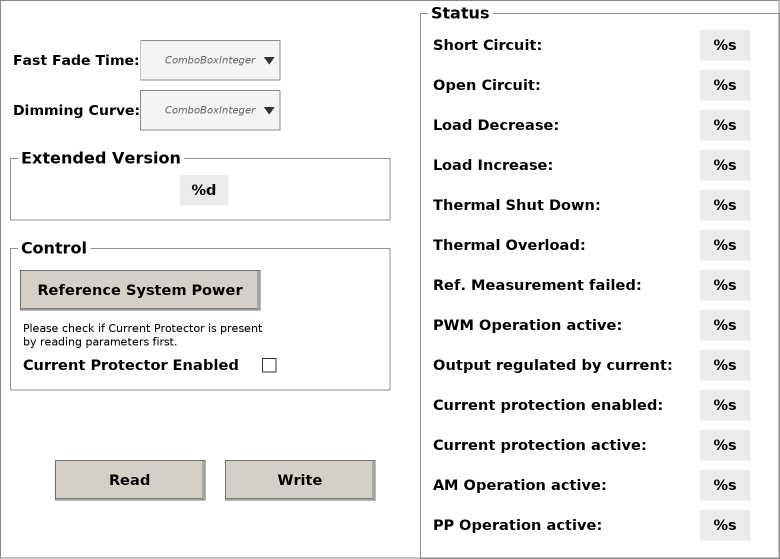
VISUALIZATION Visu_Part207Status  // 780x559
    GroupBox (420,5 360x554), "Status"
        Textfield (10,25 250x30), "Short Circuit:"
        Textfield (10,65 250x30), "Open Circuit:"
        Textfield (10,105 250x30), "Load Decrease:"
        Textfield (280,25 50x30), "%s", text variable: DALI_Commissioning.fbPart207LED.sShortCircuit
        Textfield (280,65 50x30), "%s", text variable: DALI_Commissioning.fbPart207LED.sOpenCircuit
        Textfield (280,105 50x30), "%s", text variable: DALI_Commissioning.fbPart207LED.sLoadDecrease
        Textfield (10,145 250x30), "Load Increase:"
        Textfield (280,145 50x30), "%s", text variable: DALI_Commissioning.fbPart207LED.sLoadIncrease
        Textfield (10,345 250x30), "Output regulated by current:", invisible if: DALI_Commissioning.fbPart207LED.bInvisible
        Textfield (10,385 250x30), "Current protection enabled:", invisible if: DALI_Commissioning.fbPart207LED.bInvisible
        Textfield (10,425 250x30), "Current protection active:", invisible if: DALI_Commissioning.fbPart207LED.bInvisible
        Textfield (10,185 250x30), "Thermal Shut Down:"
        Textfield (10,225 250x30), "Thermal Overload:"
        Textfield (10,265 250x30), "Ref. Measurement failed:"
        Textfield (10,465 250x30), "AM Operation active:", invisible if: DALI_Commissioning.fbPart207LED.bInvisible
        Textfield (10,505 250x30), "PP Operation active:", invisible if: DALI_Commissioning.fbPart207LED.bInvisible
        Textfield (10,305 250x30), "PWM Operation active:", invisible if: DALI_Commissioning.fbPart207LED.bInvisible
        Textfield (280,225 50x30), "%s", text variable: DALI_Commissioning.fbPart207LED.sThermalOverload
        Textfield (280,425 50x30), "%s", text variable: DALI_Commissioning.fbPart207LED.sCurrentProtectorActive, invisible if: DALI_Commissioning.fbPart207LED.bInvisible
        Textfield (280,385 50x30), "%s", text variable: DALI_Commissioning.fbPart207LED.sCurrentProtectorEnabled, invisible if: DALI_Commissioning.fbPart207LED.bInvisible
        Textfield (280,345 50x30), "%s", text variable: DALI_Commissioning.fbPart207LED.sOutputCurrentControlled, invisible if: DALI_Commissioning.fbPart207LED.bInvisible
        Textfield (280,465 50x30), "%s", text variable: DALI_Commissioning.fbPart207LED.sAMOperation, invisible if: DALI_Commissioning.fbPart207LED.bInvisible
        Textfield (280,505 50x30), "%s", text variable: DALI_Commissioning.fbPart207LED.sPowerPulseOperation, invisible if: DALI_Commissioning.fbPart207LED.bInvisible
        Textfield (280,265 50x30), "%s", text variable: DALI_Commissioning.fbPart207LED.sReferenceMeasurementFailed
        Textfield (280,185 50x30), "%s", text variable: DALI_Commissioning.fbPart207LED.sThermalShutDown
        Textfield (280,305 50x30), "%s", text variable: DALI_Commissioning.fbPart207LED.sPWMOperation, invisible if: DALI_Commissioning.fbPart207LED.bInvisible
    Button (225,460 150x40), "Write"
        OnMouseClick: execute { DALI_Commissioning.fbPart207LED.bWrite := TRUE; }
    GroupBox (10,240 380x150), "Control"
        Textfield (10,110 230x30), "Current Protector Enabled", invisible if: NOT DALI_Commissioning.fbPart207LED.bQueryCurrentProtectionDevicePresent
        Checkbox (250,110 30x30), variable: DALI_Commissioning.fbPart207LED.bCurrentProtector, invisible if: NOT DALI_Commissioning.fbPart207LED.bQueryCurrentProtectionDevicePresent, input disabled if: DALI_Commissioning.fbPart207LED.bQueryCurrentProtectionDevicePresent
        Button (10,30 240x40), "Reference System Power"
            OnMouseClick: execute { DALI_Commissioning.fbPart207LED.bReferenceSystempower := TRUE; }
        Label (10,80 300x30), "Please check if Current Protector is present by reading parameters first."
    Button (55,460 150x40), "Read"
        OnMouseClick: execute { DALI_Commissioning.fbPart207LED.bReadStatus := TRUE; }
    GroupBox (10,150 380x70), "Extended Version"
        Textfield (170,25 48x30), "%d", text variable: DALI_Commissioning.fbPart207LED.nExtendedVersionNumber
    Group (10,90 270x40)
        Textfield (0,0 130x40), "Dimming Curve:"
        ComboBoxInteger (130,0 140x40), variable: DALI_Commissioning.fbPart207LED.eDimmingCurve, text list: 'DimmingCurve'
    Group (10,40 270x40)
        ComboBoxInteger (130,0 140x40), variable: DALI_Commissioning.fbPart207LED.eFastFadeTime, text list: 'FastFadeTime'
        Textfield (0,0 130x40), "Fast Fade Time:"
END_VISUALIZATION

(* stored: Version 1.1.0.1, ProductVersion 3.1.4024.12
   Visu Visu_Part207Status: Id {3fdb9a69-24e2-43b5-83d3-017cfcbce496} *)
